// Mitsubishi GX Works2 project: 240402_우선순위회로   PLC: Q03UDV

PROGRAM MAIN
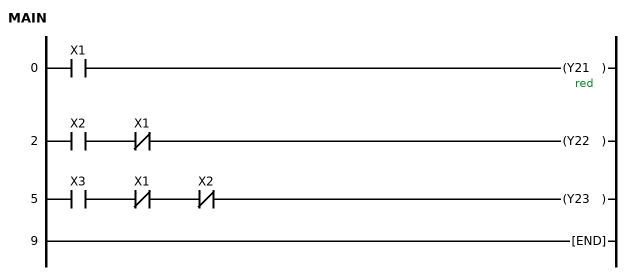
0     LD      X1
      OUT     Y21  ; red
2     LD      X2
      ANI     X1
      OUT     Y22
5     LD      X3
      ANI     X1
      ANI     X2
      OUT     Y23
9     END
END_PROGRAM
